# EPICS substitutions: lakeshore336App/Db/lakeshore336_channelnames.substitutions
file "lakeshore336_channelnames.template" {
     pattern { ChIndex }

    { A  }
    { B  }
    { C1 }
    { C2 }
    { C3 }
    { C4 }
    { C5 }
    { D1 }
    { D2 }
    { D3 }
    { D4 }
    { D5 }
}
